INTERFACE I_BaseFB EXTENDS I_InterfaceBase

PROPERTY Busy : BOOL
GET
END_GET
END_PROPERTY

PROPERTY Error : BOOL
GET
END_GET
END_PROPERTY

PROPERTY ErrorID : UDINT;
GET
END_GET
END_PROPERTY

END_INTERFACE

(* stored: Version 1.1.0.1, ProductVersion 3.1.4024.12
   Itf I_BaseFB: Id {6fd981cf-884e-4b66-abf9-487f47b0c4a4}
   Property Busy: Id {76fc170c-6eb4-4c7e-815c-66e1c0a84bb7}
   Get Get: Id {21f9484d-f357-49d2-b322-8e618b6de7c7}
   Property Error: Id {6d5e5a53-4d74-4214-bde8-c2227be1d4e0}
   Get Get: Id {28beb5b2-db14-4af2-a054-33a5fe0bc13a}
   Property ErrorID: Id {58ef2394-add9-41c0-b67b-16d4cc8fb7b0}
   Get Get: Id {6f5a0228-27d7-4baa-a925-3ff0ae6e3c19} *)
